PROGRAM PRG_07_ZAxis
VAR
	bZAxisApproachingDownLimit: BOOL;
	lSawUpLimitValue: LREAL;
	lSawDownLimitValue: LREAL;
END_VAR

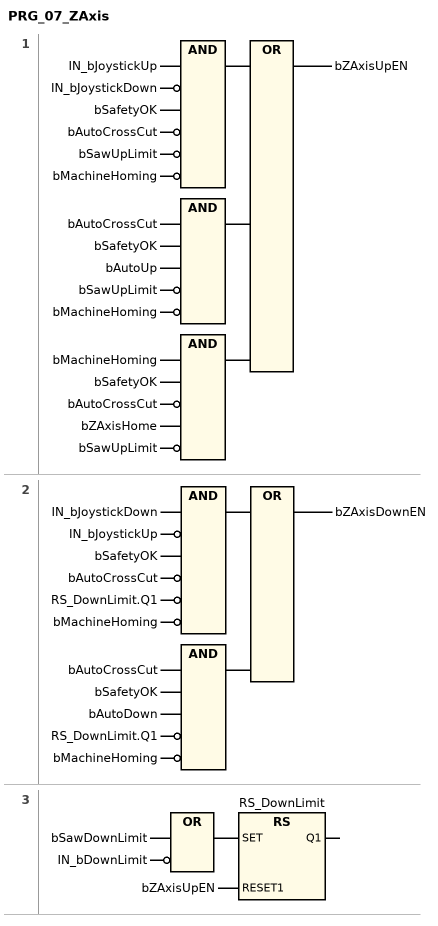
// NETWORK 1
bZAxisUpEN := IN_bJoystickUp AND NOT IN_bJoystickDown AND bSafetyOK AND NOT bAutoCrossCut AND NOT bSawUpLimit AND NOT bMachineHoming OR bAutoCrossCut AND bSafetyOK AND bAutoUp AND NOT bSawUpLimit AND NOT bMachineHoming OR bMachineHoming AND bSafetyOK AND NOT bAutoCrossCut AND bZAxisHome AND NOT bSawUpLimit;

// NETWORK 2
bZAxisDownEN := IN_bJoystickDown AND NOT IN_bJoystickUp AND bSafetyOK AND NOT bAutoCrossCut AND NOT RS_DownLimit.Q1 AND NOT bMachineHoming OR bAutoCrossCut AND bSafetyOK AND bAutoDown AND NOT RS_DownLimit.Q1 AND NOT bMachineHoming;

// NETWORK 3
RS_DownLimit(SET := bSawDownLimit OR NOT IN_bDownLimit, RESET1 := bZAxisUpEN); // RS

ACTION ACT_07_1_ZAxis:
lSawUpLimitValue := 0 ;			// Z-Axis up limit
lSawDownLimitValue := 384.50 ;	// Z-Axis down limit with 36" setup blade

GVL.Z2_Axis.AchsIn.IstPos;

//Z-Axis Up limit encoder value
IF GVL.Z2_Axis.AchsIn.IstPos >= lSawUpLimitValue THEN
	bSawUpLimit := FALSE;
ELSE bSawUpLimit := TRUE ;
END_IF

//Z-Axis Down limit encoder value
IF GVL.Z2_Axis.AchsIn.IstPos <= lSawDownLimitValue THEN
	bSawDownLimit := FALSE;
ELSE bSawDownLimit := TRUE;
END_IF

// Z-Axis Approaching down limit
IF GVL.Z2_Axis.AchsIn.IstPos >= lSawDownLimitValue - 35 THEN
	bZAxisApproachingDownLimit := TRUE ;
ELSE bZAxisApproachingDownLimit := FALSE ;
END_IF

// Z-Axis Speed
IF bZAxisApproachingDownLimit AND bZAxisDownEN THEN
	rZAxisSpeed := 5 ;
ELSE rZAxisSpeed := 25;
END_IF

// Z-Axis Down limit redundancy in case inductive sensor fails



// AutoCrossCut double pass reference
END_ACTION

END_PROGRAM

(* stored: Version 1.1.0.1, ProductVersion 3.1.4024.15
   POU PRG_07_ZAxis: Id {12ac2dd4-f6da-4ca8-a1c9-34a1b40bca30}, SpecialFunc None
   Action ACT_07_1_ZAxis: Id {37eede63-3491-4d39-819a-d0a9e71862d9} *)
